INTERFACE I_Deserializable EXTENDS __SYSTEM.IQueryInterface

METHOD TryDeserializeFrom : BOOL
VAR_INPUT
	Deserializer : I_Deserializer;
	Feedback : I_DeserializerFeedback;
END_VAR
END_METHOD

END_INTERFACE

(* stored: Version 1.1.0.1, ProductVersion 3.1.4024.12
   Itf I_Deserializable: Id {304c5669-cf3c-09f7-0c3a-89b35734a234}
   Method TryDeserializeFrom: Id {33ef4acc-db66-0b4b-21c5-3d5be6a2e887} *)
